(* Ange vilken datumarray som är aktuell beroende på aktuellt år *)
IF _uiYY=2017
THEN AktuellDatumArray:=Array2017;
ELSIF _uiYY=2018
THEN AktuellDatumArray:=Array2018;
ELSIF _uiYY=2019
THEN AktuellDatumArray:=Array2019;
ELSIF _uiYY=2020
THEN AktuellDatumArray:=Array2020;
ELSIF _uiYY=2021
THEN AktuellDatumArray:=Array2021;
ELSIF _uiYY=2022
THEN AktuellDatumArray:=Array2022;
ELSIF _uiYY=2023
THEN AktuellDatumArray:=Array2023;
ELSIF _uiYY=2024
THEN AktuellDatumArray:=Array2024;
ELSIF _uiYY=2025
THEN AktuellDatumArray:=Array2025;
ELSIF _uiYY=2026
THEN AktuellDatumArray:=Array2026;
ELSIF _uiYY=2027
THEN AktuellDatumArray:=Array2027;
ELSIF _uiYY=2028
THEN AktuellDatumArray:=Array2028;
ELSIF _uiYY=2029
THEN AktuellDatumArray:=Array2029;
ELSIF _uiYY=2030
THEN AktuellDatumArray:=Array2030;
ELSIF _uiYY=2031
THEN AktuellDatumArray:=Array2031;
ELSIF _uiYY=2032
THEN AktuellDatumArray:=Array2032;
ELSIF _uiYY=2033
THEN AktuellDatumArray:=Array2033;
ELSIF _uiYY=2034
THEN AktuellDatumArray:=Array2034;
ELSIF _uiYY=2035
THEN AktuellDatumArray:=Array2035;
ELSIF _uiYY=2036
THEN AktuellDatumArray:=Array2036;
ELSIF _uiYY=2037
THEN AktuellDatumArray:=Array2037;
END_IF


(* Kolla om dagens datum stämmer överens med någon av inställda helgdagar/-aftnar*)
IF _rDatum=AktuellDatumArray[1]			(*Trettondagsafton*)
OR _rDatum= AktuellDatumArray[2]			(*Skartorsdag*)
OR _rDatum=AktuellDatumArray[3]			(*Paskafton*)
OR _rDatum=AktuellDatumArray[4]			(*Valborgsmassoafton*)
OR _rDatum=AktuellDatumArray[5]			(*Pingstafton*)
OR _rDatum=AktuellDatumArray[6]			(*Midsommarafton*)
OR _rDatum=AktuellDatumArray[7]			(*AllaHelgonsAfton*)
OR _rDatum=AktuellDatumArray[8]			(*Julafton*)
OR _rDatum=AktuellDatumArray[9]			(*Nyarsafton*)
THEN bDFH:=TRUE;
ELSE bDFH:=FALSE;
END_IF

IF _rDatum=AktuellDatumArray[10]			(*Nyarsdagen*)
OR _rDatum=AktuellDatumArray[11]			(*TrettondagJul*)
OR _rDatum=AktuellDatumArray[12]			(*Langfredag*)
OR _rDatum=AktuellDatumArray[13]			(*Paskdagen*)
OR _rDatum=AktuellDatumArray[14]			(*AnnandagPask*)
OR _rDatum=AktuellDatumArray[15]			(*ForstaMaj*)
OR _rDatum=AktuellDatumArray[16]			(*KristiHimmelsfard*)
OR _rDatum=AktuellDatumArray[17]			(*Pingstdagen*)
OR _rDatum=AktuellDatumArray[18]			(*Nationaldagen*)
OR _rDatum=AktuellDatumArray[19]			(*Midsommardagen*)
OR _rDatum=AktuellDatumArray[20]			(*AllaHelgonsDag*)
OR _rDatum=AktuellDatumArray[21]			(*Juldagen*)
OR _rDatum=AktuellDatumArray[22]			(*AnnandagJul*)
THEN bHD:=TRUE;
ELSE bHD:=FALSE;
END_IF


(*Sätt larmutgång till TRUE om aktuellt årtal är större än 2037*)
IF  _uiYY>2037
THEN bLarm:=TRUE;
ELSE bLarm:=FALSE;
END_IF
END_FUNCTION_BLOCK

(* POU SYSTEM/HUS2_AS01_GT3N, CFC *)
PROGRAM HUS2_AS01_GT3N
VAR

	FilterDelay: fbDelayedAlarmMinutes;
END_VAR
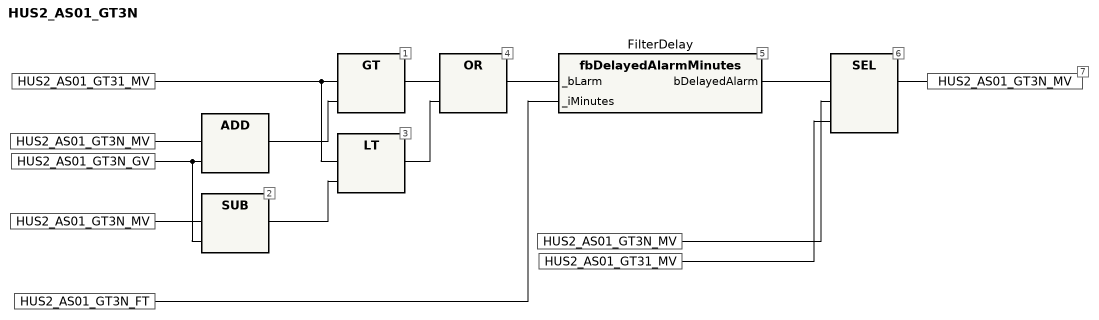
_CFC_ (* Continuous Function Chart, elements in execution order *)
#0 ADD(HUS2_AS01_GT3N_MV, HUS2_AS01_GT3N_GV)
#1 GT(HUS2_AS01_GT31_MV, #0)
#2 SUB(HUS2_AS01_GT3N_MV, HUS2_AS01_GT3N_GV)
#3 LT(HUS2_AS01_GT31_MV, #2)
#4 OR(#1, #3)
#5 FilterDelay:fbDelayedAlarmMinutes(_bLarm: #4, _iMinutes: HUS2_AS01_GT3N_FT)
#6 SEL(#5.bDelayedAlarm, HUS2_AS01_GT3N_MV, HUS2_AS01_GT31_MV)
#7 HUS2_AS01_GT3N_MV <= #6
_END_CFC_
(* the same logic as Structured Text *)
FilterDelay(_bLarm := (HUS2_AS01_GT31_MV > (HUS2_AS01_GT3N_MV + HUS2_AS01_GT3N_GV)) OR (HUS2_AS01_GT31_MV < (HUS2_AS01_GT3N_MV - HUS2_AS01_GT3N_GV)), _iMinutes := HUS2_AS01_GT3N_FT);
HUS2_AS01_GT3N_MV := SEL(FilterDelay.bDelayedAlarm, HUS2_AS01_GT3N_MV, HUS2_AS01_GT31_MV);
END_PROGRAM

(* POU SYSTEM/HUS2_AS01_SOMMARVINTER, CFC *)
PROGRAM HUS2_AS01_SOMMARVINTER

VAR
	udiIntval      : UDINT:=3600;
	udiNumOfElem   : UDINT:=72;
	lrOut             : LREAL;
	lrMax             : LREAL;
	lrMin             : LREAL;
	udiStaNumOfElem   : UDINT;

	AverageCalc: FB_HVACTimeAverage;
	ActivationDelay: TON;

	SetReset: SR;
	bVINTER_TILL: BOOL;
	TEST: BOOL := TRUE;
	TFD_VINTER: TON;
	TFD_DELAY_BER: fbINT_TO_MIN;
	FFD_VINTER: TON;
	FFD_DELAY_BER: fbINT_TO_MIN;
END_VAR
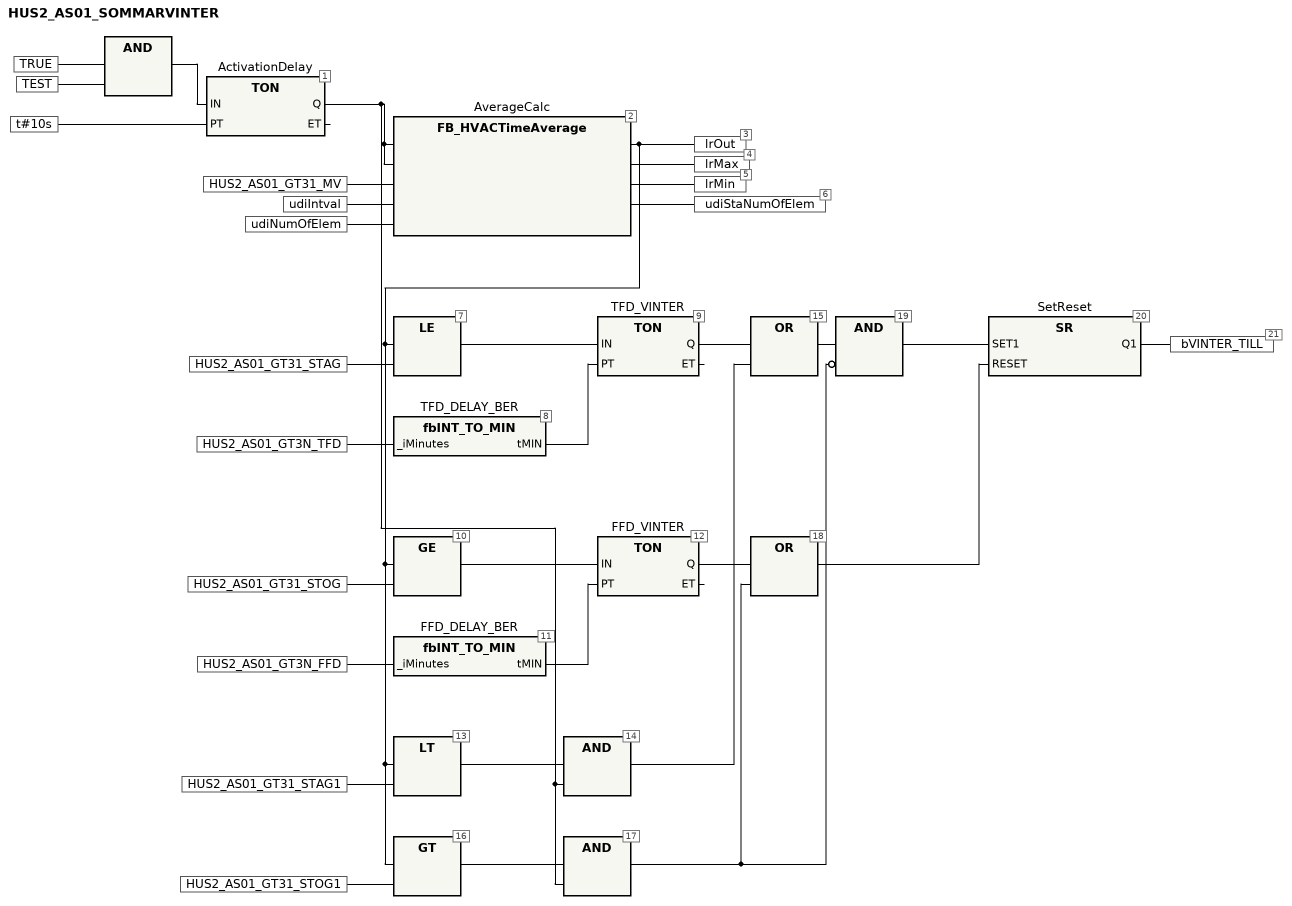
_CFC_ (* Continuous Function Chart, elements in execution order *)
#0 AND(TRUE, TEST)
#1 ActivationDelay:TON(IN: #0, PT: t#10s)
#2 AverageCalc:FB_HVACTimeAverage(#1.Q, #1.Q, HUS2_AS01_GT31_MV, udiIntval, udiNumOfElem)
#3 lrOut <= #2.out 1
#4 lrMax <= #2.out 2
#5 lrMin <= #2.out 3
#6 udiStaNumOfElem <= #2.out 4
#7 LE(#2.out 1, HUS2_AS01_GT31_STAG)
#8 TFD_DELAY_BER:fbINT_TO_MIN(_iMinutes: HUS2_AS01_GT3N_TFD)
#9 TFD_VINTER:TON(IN: #7, PT: #8.tMIN)
#10 GE(#2.out 1, HUS2_AS01_GT31_STOG)
#11 FFD_DELAY_BER:fbINT_TO_MIN(_iMinutes: HUS2_AS01_GT3N_FFD)
#12 FFD_VINTER:TON(IN: #10, PT: #11.tMIN)
#13 LT(#2.out 1, HUS2_AS01_GT31_STAG1)
#14 AND(#13, #1.Q)
#15 OR(#9.Q, #14)
#16 GT(#2.out 1, HUS2_AS01_GT31_STOG1)
#17 AND(#16, #1.Q)
#18 OR(#12.Q, #17)
#19 AND(#15, NOT #17)
#20 SetReset:SR(SET1: #19, RESET: #18)
#21 bVINTER_TILL <= #20.Q1
_END_CFC_
END_PROGRAM

(* POU xEgna Funktionsblock/fbINT_TO_MIN, CFC *)
FUNCTION_BLOCK fbINT_TO_MIN
VAR_INPUT
	_iMinutes  :INT;
END_VAR

VAR_OUTPUT
	tMIN: TIME;
END_VAR
VAR (* helpers for the ST form of the networks *)
	_t10 : TIME;
END_VAR
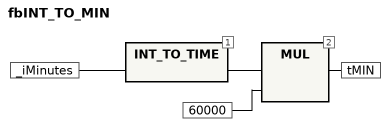
_CFC_ (* Continuous Function Chart, elements in execution order *)
#0 tMIN <= #2
#1 INT_TO_TIME(_iMinutes)
#2 MUL(#1, 60000)
_END_CFC_
(* the same logic as Structured Text *)
tMIN := _t10;
_t10 := INT_TO_TIME(_iMinutes) * 60000;
END_FUNCTION_BLOCK

(* POU SYSTEM/HUS2_AS01_LARMLAMPA, CFC *)
PROGRAM HUS2_AS01_LARMLAMPA
VAR

	BLINKALARM: FB_HVACBlink;
	ResetSet: RS;
	ACK: BOOL;
	TRIG1: R_TRIG;

	WEBPORT: BOOL;
	RESET_ACK: fbBool_Reset;
END_VAR
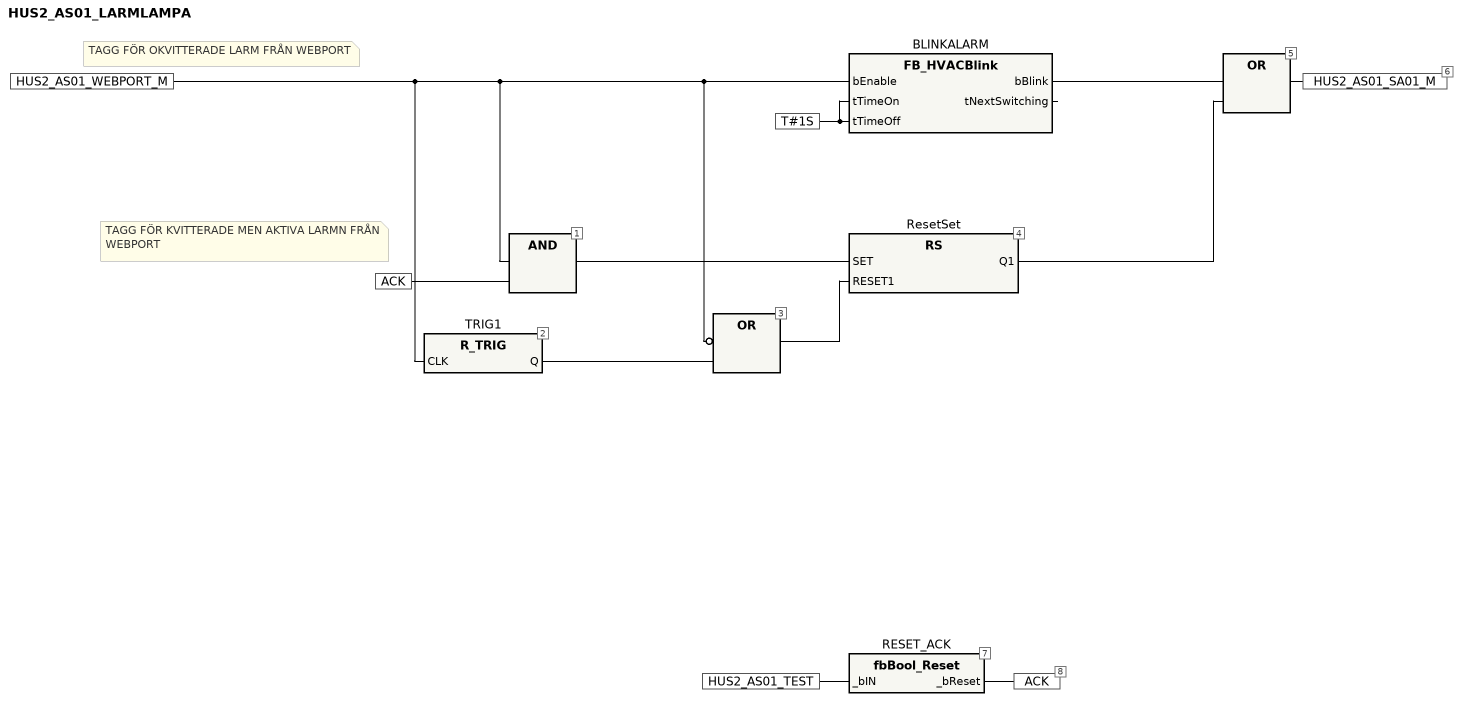
_CFC_ (* Continuous Function Chart, elements in execution order *)
(* TAGG FÖR OKVITTERADE LARM FRÅN WEBPORT *)
#0 BLINKALARM:FB_HVACBlink(bEnable: HUS2_AS01_WEBPORT_M, tTimeOn: T#1S, tTimeOff: T#1S)
#1 AND(HUS2_AS01_WEBPORT_M, ACK)
#2 TRIG1:R_TRIG(CLK: HUS2_AS01_WEBPORT_M)
#3 OR(NOT HUS2_AS01_WEBPORT_M, #2.Q)
#4 ResetSet:RS(SET: #1, RESET1: #3)
#5 OR(#0.bBlink, #4.Q1)
#6 HUS2_AS01_SA01_M <= #5
#7 RESET_ACK:fbBool_Reset(_bIN: HUS2_AS01_TEST)
#8 ACK <= #7._bReset
(* TAGG FÖR KVITTERADE MEN AKTIVA LARMN FRÅN WEBPORT *)
_END_CFC_
(* the same logic as Structured Text *)
(* TAGG FÖR OKVITTERADE LARM FRÅN WEBPORT *)
BLINKALARM(bEnable := HUS2_AS01_WEBPORT_M, tTimeOn := T#1S, tTimeOff := T#1S);
TRIG1(CLK := HUS2_AS01_WEBPORT_M);
ResetSet(SET := HUS2_AS01_WEBPORT_M AND ACK, RESET1 := NOT HUS2_AS01_WEBPORT_M OR TRIG1.Q);
HUS2_AS01_SA01_M := BLINKALARM.bBlink OR ResetSet.Q1;
RESET_ACK(_bIN := HUS2_AS01_TEST);
ACK := RESET_ACK._bReset;
(* TAGG FÖR KVITTERADE MEN AKTIVA LARMN FRÅN WEBPORT *)
END_PROGRAM

(* POU SYSTEM/Belysning/HUS2_AS01_Belysning_MAIN, CFC *)
PROGRAM HUS2_AS01_Belysning_MAIN
VAR
	LUXSTYR_BE01: fbLUX_ON_OFF;
	LUXSTYR_BE02: fbLUX_ON_OFF;
END_VAR
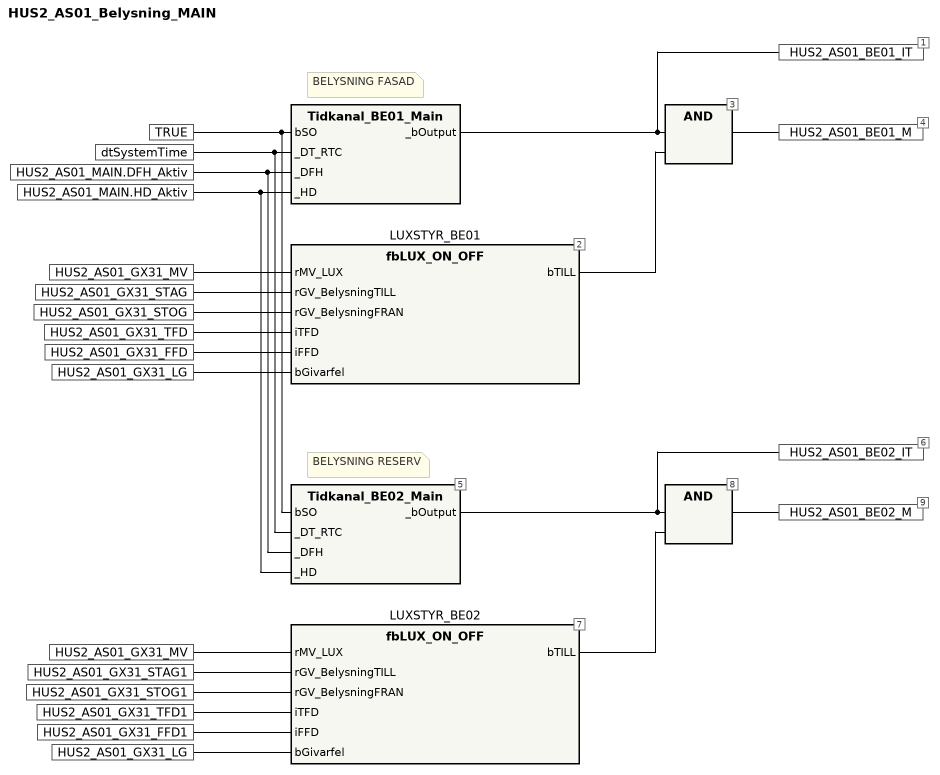
_CFC_ (* Continuous Function Chart, elements in execution order *)
(* BELYSNING FASAD *)
(* BELYSNING RESERV *)
#0 Tidkanal_BE01_Main(bSO: TRUE, _DT_RTC: dtSystemTime, _DFH: HUS2_AS01_MAIN.DFH_Aktiv, _HD: HUS2_AS01_MAIN.HD_Aktiv)
#1 HUS2_AS01_BE01_IT <= #0._bOutput
#2 LUXSTYR_BE01:fbLUX_ON_OFF(rMV_LUX: HUS2_AS01_GX31_MV, rGV_BelysningTILL: HUS2_AS01_GX31_STAG, rGV_BelysningFRAN: HUS2_AS01_GX31_STOG, iTFD: HUS2_AS01_GX31_TFD, iFFD: HUS2_AS01_GX31_FFD, bGivarfel: HUS2_AS01_GX31_LG)
#3 AND(#0._bOutput, #2.bTILL)
#4 HUS2_AS01_BE01_M <= #3
#5 Tidkanal_BE02_Main(bSO: TRUE, _DT_RTC: dtSystemTime, _DFH: HUS2_AS01_MAIN.DFH_Aktiv, _HD: HUS2_AS01_MAIN.HD_Aktiv)
#6 HUS2_AS01_BE02_IT <= #5._bOutput
#7 LUXSTYR_BE02:fbLUX_ON_OFF(rMV_LUX: HUS2_AS01_GX31_MV, rGV_BelysningTILL: HUS2_AS01_GX31_STAG1, rGV_BelysningFRAN: HUS2_AS01_GX31_STOG1, iTFD: HUS2_AS01_GX31_TFD1, iFFD: HUS2_AS01_GX31_FFD1, bGivarfel: HUS2_AS01_GX31_LG)
#8 AND(#5._bOutput, #7.bTILL)
#9 HUS2_AS01_BE02_M <= #8
_END_CFC_
(* the same logic as Structured Text *)
(* BELYSNING FASAD *)
(* BELYSNING RESERV *)
Tidkanal_BE01_Main(bSO := TRUE, _DT_RTC := dtSystemTime, _DFH := HUS2_AS01_MAIN.DFH_Aktiv, _HD := HUS2_AS01_MAIN.HD_Aktiv);
HUS2_AS01_BE01_IT := Tidkanal_BE01_Main._bOutput;
LUXSTYR_BE01(rMV_LUX := HUS2_AS01_GX31_MV, rGV_BelysningTILL := HUS2_AS01_GX31_STAG, rGV_BelysningFRAN := HUS2_AS01_GX31_STOG, iTFD := HUS2_AS01_GX31_TFD, iFFD := HUS2_AS01_GX31_FFD, bGivarfel := HUS2_AS01_GX31_LG);
HUS2_AS01_BE01_M := Tidkanal_BE01_Main._bOutput AND LUXSTYR_BE01.bTILL;
Tidkanal_BE02_Main(bSO := TRUE, _DT_RTC := dtSystemTime, _DFH := HUS2_AS01_MAIN.DFH_Aktiv, _HD := HUS2_AS01_MAIN.HD_Aktiv);
HUS2_AS01_BE02_IT := Tidkanal_BE02_Main._bOutput;
LUXSTYR_BE02(rMV_LUX := HUS2_AS01_GX31_MV, rGV_BelysningTILL := HUS2_AS01_GX31_STAG1, rGV_BelysningFRAN := HUS2_AS01_GX31_STOG1, iTFD := HUS2_AS01_GX31_TFD1, iFFD := HUS2_AS01_GX31_FFD1, bGivarfel := HUS2_AS01_GX31_LG);
HUS2_AS01_BE02_M := Tidkanal_BE02_Main._bOutput AND LUXSTYR_BE02.bTILL;
END_PROGRAM

(* POU xEgna Funktionsblock/fbLUX_ON_OFF, CFC *)
FUNCTION_BLOCK fbLUX_ON_OFF

VAR_INPUT
	rMV_LUX					: REAL;
	rGV_BelysningTILL		: REAL;
	rGV_BelysningFRAN		: REAL;
	iTFD						: INT;
	iFFD						: INT;
	bGivarfel					: BOOL;
END_VAR
VAR
	DelayON: TON;
	DelayOFF: TON;
	SETRESET: SR;
END_VAR
VAR_OUTPUT
	bTILL: BOOL;
END_VAR
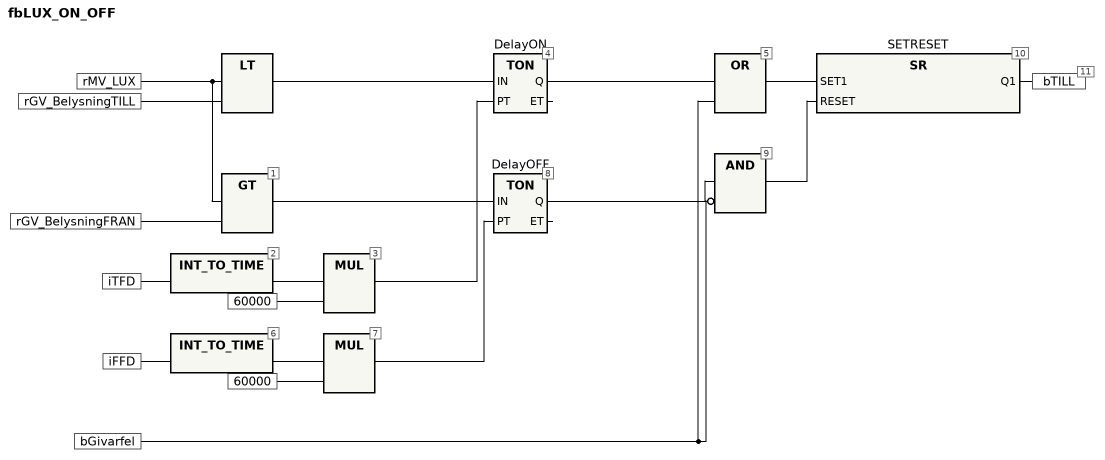
_CFC_ (* Continuous Function Chart, elements in execution order *)
#0 LT(rMV_LUX, rGV_BelysningTILL)
#1 GT(rMV_LUX, rGV_BelysningFRAN)
#2 INT_TO_TIME(iTFD)
#3 MUL(#2, 60000)
#4 DelayON:TON(IN: #0, PT: #3)
#5 OR(#4.Q, bGivarfel)
#6 INT_TO_TIME(iFFD)
#7 MUL(#6, 60000)
#8 DelayOFF:TON(IN: #1, PT: #7)
#9 AND(#8.Q, NOT bGivarfel)
#10 SETRESET:SR(SET1: #5, RESET: #9)
#11 bTILL <= #10.Q1
_END_CFC_
(* the same logic as Structured Text *)
DelayON(IN := rMV_LUX < rGV_BelysningTILL, PT := INT_TO_TIME(iTFD) * 60000);
DelayOFF(IN := rMV_LUX > rGV_BelysningFRAN, PT := INT_TO_TIME(iFFD) * 60000);
SETRESET(SET1 := DelayON.Q OR bGivarfel, RESET := DelayOFF.Q AND NOT bGivarfel);
bTILL := SETRESET.Q1;
END_FUNCTION_BLOCK

(* POU SYSTEM/Belysning/BE01/Tidkanal_BE01_Main, CFC *)
PROGRAM Tidkanal_BE01_Main

VAR_INPUT
	bSO: BOOL;
	_DT_RTC	:DT;
	_DFH :BOOL;
	_HD:BOOL;

END_VAR


VAR
	AUTO_MAN: fbManualOverride;

	OffDelayTK: TOF;
END_VAR

VAR_OUTPUT
	_bOutput:BOOL;

END_VAR
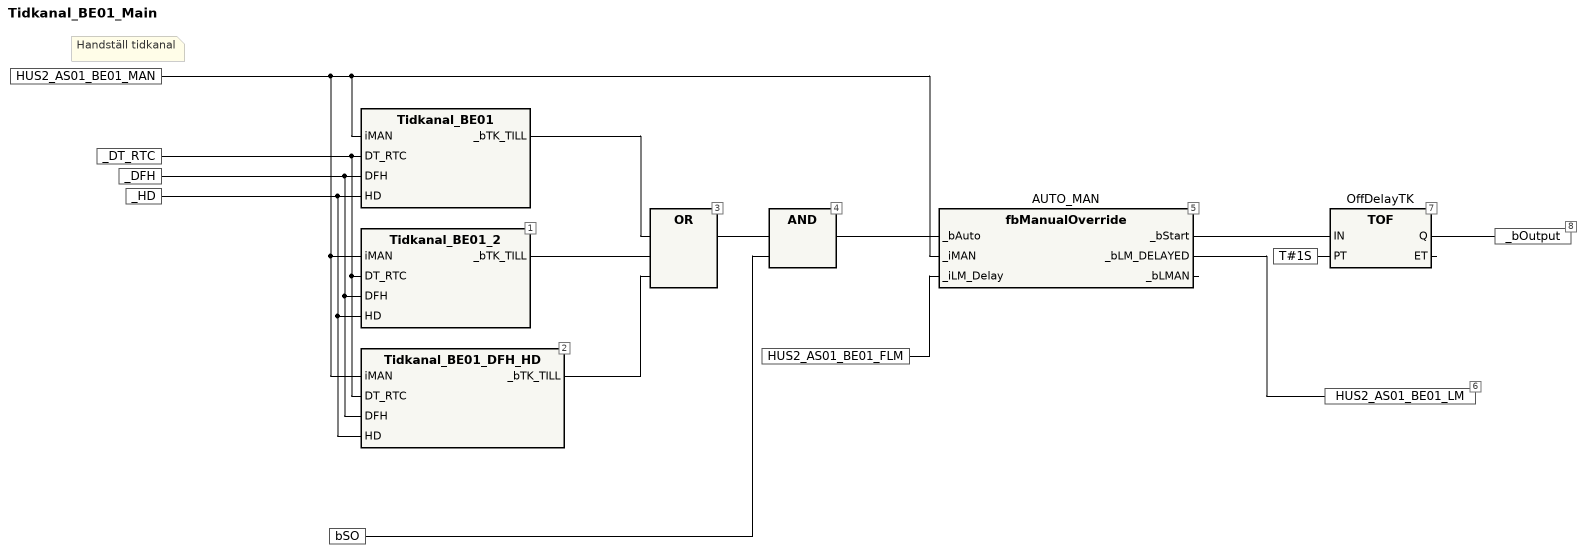
_CFC_ (* Continuous Function Chart, elements in execution order *)
(* Handställ tidkanal *)
#0 Tidkanal_BE01(iMAN: HUS2_AS01_BE01_MAN, DT_RTC: _DT_RTC, DFH: _DFH, HD: _HD)
#1 Tidkanal_BE01_2(iMAN: HUS2_AS01_BE01_MAN, DT_RTC: _DT_RTC, DFH: _DFH, HD: _HD)
#2 Tidkanal_BE01_DFH_HD(iMAN: HUS2_AS01_BE01_MAN, DT_RTC: _DT_RTC, DFH: _DFH, HD: _HD)
#3 OR(#0._bTK_TILL, #1._bTK_TILL, #2._bTK_TILL)
#4 AND(#3, bSO)
#5 AUTO_MAN:fbManualOverride(_bAuto: #4, _iMAN: HUS2_AS01_BE01_MAN, _iLM_Delay: HUS2_AS01_BE01_FLM)
#6 HUS2_AS01_BE01_LM <= #5._bLM_DELAYED
#7 OffDelayTK:TOF(IN: #5._bStart, PT: T#1S)
#8 _bOutput <= #7.Q
_END_CFC_
(* the same logic as Structured Text *)
(* Handställ tidkanal *)
Tidkanal_BE01(iMAN := HUS2_AS01_BE01_MAN, DT_RTC := _DT_RTC, DFH := _DFH, HD := _HD);
Tidkanal_BE01_2(iMAN := HUS2_AS01_BE01_MAN, DT_RTC := _DT_RTC, DFH := _DFH, HD := _HD);
Tidkanal_BE01_DFH_HD(iMAN := HUS2_AS01_BE01_MAN, DT_RTC := _DT_RTC, DFH := _DFH, HD := _HD);
AUTO_MAN(_bAuto := (Tidkanal_BE01._bTK_TILL OR Tidkanal_BE01_2._bTK_TILL OR Tidkanal_BE01_DFH_HD._bTK_TILL) AND bSO, _iMAN := HUS2_AS01_BE01_MAN, _iLM_Delay := HUS2_AS01_BE01_FLM);
HUS2_AS01_BE01_LM := AUTO_MAN._bLM_DELAYED;
OffDelayTK(IN := AUTO_MAN._bStart, PT := T#1S);
_bOutput := OffDelayTK.Q;
END_PROGRAM

(* POU xEgna Funktionsblock/fbManualOverride, CFC *)
FUNCTION_BLOCK fbManualOverride
VAR_INPUT
	_bAuto:BOOL;
	_iMAN: INT;
	_iLM_Delay: INT;
END_VAR
VAR_OUTPUT
	_bStart: BOOL;
	_bLM_DELAYED: BOOL;
	_bLMAN: BOOL;
END_VAR
VAR
	LM_DELAY: fbDelayedAlarmMinutes;
	OFF_DELAY: TOF;
END_VAR
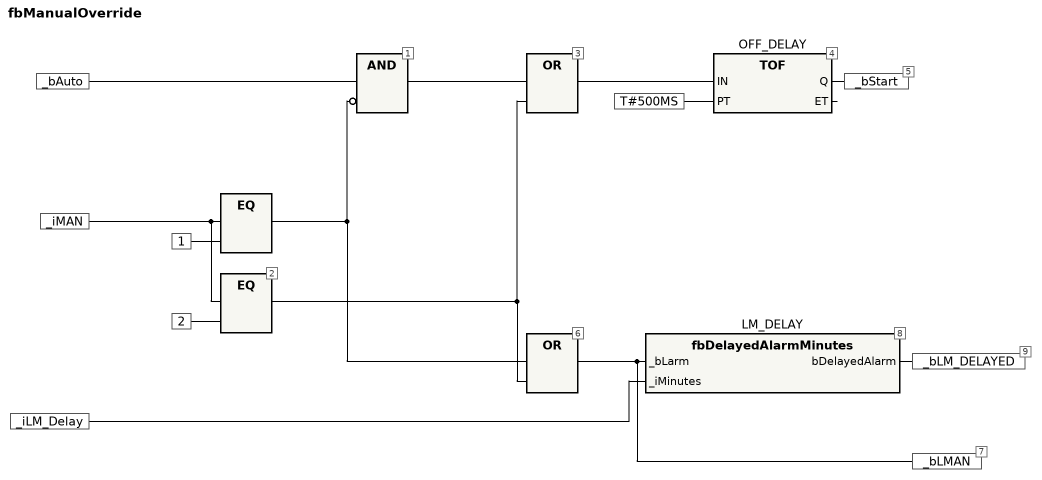
_CFC_ (* Continuous Function Chart, elements in execution order *)
#0 EQ(_iMAN, 1)
#1 AND(_bAuto, NOT #0)
#2 EQ(_iMAN, 2)
#3 OR(#1, #2)
#4 OFF_DELAY:TOF(IN: #3, PT: T#500MS)
#5 _bStart <= #4.Q
#6 OR(#0, #2)
#7 _bLMAN <= #6
#8 LM_DELAY:fbDelayedAlarmMinutes(_bLarm: #6, _iMinutes: _iLM_Delay)
#9 _bLM_DELAYED <= #8.bDelayedAlarm
_END_CFC_
(* the same logic as Structured Text *)
OFF_DELAY(IN := (_bAuto AND NOT (_iMAN = 1)) OR (_iMAN = 2), PT := T#500MS);
_bStart := OFF_DELAY.Q;
_bLMAN := (_iMAN = 1) OR (_iMAN = 2);
LM_DELAY(_bLarm := (_iMAN = 1) OR (_iMAN = 2), _iMinutes := _iLM_Delay);
_bLM_DELAYED := LM_DELAY.bDelayedAlarm;
END_FUNCTION_BLOCK

(* POU SYSTEM/Belysning/BE01/Tidkanal_BE01, FAI *)
PROGRAM Tidkanal_BE01

VAR

(****************************************  weekly time switch *********************************************************************************************************************)
	fbWeeklyTimeSwitch		:FB_HVACScheduler7ch;
	_eDST					:E_HVACDataSecurityType :=1;
	SetDefaultTimeSwitch: BOOL := FALSE;
	_uiOffsetBefore			:UINT;  (* the switch-on time is brought forward by this number of minutes *)
	_arrTimeChannel 			:ARRAY[1..7] OF ST_HVACTimeChannel;(*
							    ST_HVACTimeChannel :
							    uiOn_hh			: UINT;
							    uiOn_mm		: UINT;
							    uiOn_ss			: UINT;
							    uiOff_hh			: UINT; 
							    uiOff_mm			: UINT;
							    uiOff_ss			: UINT;
							    bEnable			: BOOL;
							    bAllDays			: BOOL;
							    bMonday			: BOOL;
							    bTuesday		: BOOL;
							    bWednesday		: BOOL;
							    bThursday		: BOOL;
							    bFriday			: BOOL;
							    bSaturday		: BOOL;
							    bSunday			: BOOL;
							    bResetAfterOn	: BOOL;
							    bQ				: BOOL; *)

	_bWeeklyClock_EdgeOn		:BOOL;(* Is TRUE for one PLC cycle after bOutput switches on *)
	_bWeeklyClock_EdgeOff		:BOOL;(* Is TRUE for one PLC cycle after bOutput switches off *)
	_tWeeklyTime_NextOn		:TIME;(* Time until the next switch-on of the time switch program. Maximum value 10080 minutes (1 week) *)
	_tWeeklyTime_NextOff		:TIME;(* Time until the next switch-off of the time switch program. Maximum forecast until midnight *)
	_bWeeklyTime_FP			:BOOL;(* fault parameter recognized *)



	_bReset_Local				:BOOL;
	_bSetDefault_Local: BOOL;

	fbSCADATime1:		FB_TimeToSCADA_1_0;
	fbSCADATime2:		FB_TimeToSCADA_1_0;
	fbSCADATime3:		FB_TimeToSCADA_1_0;
	fbSCADATime4:		FB_TimeToSCADA_1_0;
	fbSCADATime5:		FB_TimeToSCADA_1_0;
	fbSCADATime6:		FB_TimeToSCADA_1_0;
	fbSCADATime7:		FB_TimeToSCADA_1_0;






END_VAR


VAR_INPUT
	iMAN				:INT;
	DT_RTC			:DT;
	DFH 				:BOOL;
	HD					:BOOL;

END_VAR

VAR_OUTPUT
	_bTK_TILL		:BOOL;

END_VAR
(* body not read: cfc101 *)
END_PROGRAM

(* POU xEgna Funktionsblock/Time_to_SCADA/FB_TimeToSCADA_1_0, ST *)
(*
Lib: TCHVAC.LIB
*)

FUNCTION_BLOCK FB_TimeToSCADA_1_0

VAR_INPUT
END_VAR

VAR_IN_OUT
	_iCitect_OnTime:		INT;		(*Time On from HMI*)
	_iCitect_OffTime:		INT;		(*Time Off from HMI*)
END_VAR
VAR_OUTPUT
	_uiOnTime_hh:		UINT;		(*Hours for on time*)
	_uiOnTime_mm:		UINT;		(*Minutes for on time*)
	_uiOffTime_hh:		UINT;		(*Hours for off time*)
	_uiOffTime_mm:		UINT;		(*Minutes for off time*)
	_bEnableTimeCh:		BOOL;		(*Enable timechannel*)
END_VAR
VAR
	iNowOn:				INT;		(*Temp var for on time*)
	iNowOff:				INT;		(*Temp var for off time*)
	fbSaveOnTime:		FB_HVACPersistent_Int;
	fbSaveOffTime:		FB_HVACPersistent_Int;
END_VAR

(*
	This FB converts hmi time from Citect to HVAC TimeChannel
	the input time is an integer. i.e Time 15:46 = _iCitect_OnTime 1546. Then
	the our and minute is extracted to the HVAC time. 
	No error handling if time is not in the appropriate range.
	Maybe the persistent data handling for the TC needs to be disabled
*)
(*Find out if we have some time set, then enable the output*)
IF
_iCitect_OffTime <> _iCitect_OnTime
THEN
(*Get the on time*)
iNowOn := _iCitect_OnTime;
(*Get hour*)
_uiOnTime_hh := iNowOn / 100;
(*Get minute*)
_uiOnTime_mm := iNowOn - ( _uiOnTime_hh * 100);

(*Get the off time*)
iNowOff := _iCitect_OffTime;
(*Get hour*)
_uiOffTime_hh := iNowOff / 100;
(*Get minute*)
_uiOffTime_mm := iNowOff - ( _uiOffTime_hh * 100);
	_bEnableTimeCh := TRUE;
ELSIF
_iCitect_OffTime=2359 AND _iCitect_OnTime=2359
OR
_iCitect_OffTime=2400 AND _iCitect_OnTime=0000
THEN
	_uiOnTime_hh:=0;
	_uiOnTime_mm:=0;
	_uiOffTime_hh:=0;
	_uiOffTime_mm:=0;
	_bEnableTimeCh:=0;
	_bEnableTimeCh := TRUE;
ELSE
	_bEnableTimeCh := FALSE;
END_IF


(*Save the on/off time data persistent*)
fbSaveOnTime(bSetDefault:= , iVar_Default:= , iVar:= _iCitect_OnTime );
fbSaveOffTime(bSetDefault:= , iVar_Default:= , iVar:= _iCitect_OffTime );
END_FUNCTION_BLOCK

(* POU SYSTEM/Belysning/BE01/Tidkanal_BE01_2, FAI *)
PROGRAM Tidkanal_BE01_2

VAR

(****************************************  weekly time switch *********************************************************************************************************************)
	fbWeeklyTimeSwitch		:FB_HVACScheduler7ch;
	_eDST					:E_HVACDataSecurityType :=1;
	SetDefaultTimeSwitch: BOOL := FALSE;
	_uiOffsetBefore			:UINT;  (* the switch-on time is brought forward by this number of minutes *)
	_arrTimeChannel 			:ARRAY[1..7] OF ST_HVACTimeChannel;(*
							    ST_HVACTimeChannel :
							    uiOn_hh			: UINT;
							    uiOn_mm		: UINT;
							    uiOn_ss			: UINT;
							    uiOff_hh			: UINT; 
							    uiOff_mm			: UINT;
							    uiOff_ss			: UINT;
							    bEnable			: BOOL;
							    bAllDays			: BOOL;
							    bMonday			: BOOL;
							    bTuesday		: BOOL;
							    bWednesday		: BOOL;
							    bThursday		: BOOL;
							    bFriday			: BOOL;
							    bSaturday		: BOOL;
							    bSunday			: BOOL;
							    bResetAfterOn	: BOOL;
							    bQ				: BOOL; *)

	_bWeeklyClock_EdgeOn		:BOOL;(* Is TRUE for one PLC cycle after bOutput switches on *)
	_bWeeklyClock_EdgeOff		:BOOL;(* Is TRUE for one PLC cycle after bOutput switches off *)
	_tWeeklyTime_NextOn		:TIME;(* Time until the next switch-on of the time switch program. Maximum value 10080 minutes (1 week) *)
	_tWeeklyTime_NextOff		:TIME;(* Time until the next switch-off of the time switch program. Maximum forecast until midnight *)
	_bWeeklyTime_FP			:BOOL;(* fault parameter recognized *)



	_bReset_Local				:BOOL;
	_bSetDefault_Local: BOOL;

	fbSCADATime1:		FB_TimeToSCADA_1_0;
	fbSCADATime2:		FB_TimeToSCADA_1_0;
	fbSCADATime3:		FB_TimeToSCADA_1_0;
	fbSCADATime4:		FB_TimeToSCADA_1_0;
	fbSCADATime5:		FB_TimeToSCADA_1_0;
	fbSCADATime6:		FB_TimeToSCADA_1_0;
	fbSCADATime7:		FB_TimeToSCADA_1_0;






END_VAR


VAR_INPUT
	iMAN				:INT;
	DT_RTC			:DT;
	DFH 				:BOOL;
	HD					:BOOL;

END_VAR

VAR_OUTPUT
	_bTK_TILL		:BOOL;

END_VAR
(* body not read: cfc101 *)
END_PROGRAM

(* POU SYSTEM/Belysning/BE01/Tidkanal_BE01_DFH_HD, FAI *)
PROGRAM Tidkanal_BE01_DFH_HD

VAR

(****************************************  weekly time switch *********************************************************************************************************************)
	fbWeeklyTimeSwitch		:FB_HVACScheduler7ch;
	_eDST					:E_HVACDataSecurityType :=1;
	SetDefaultTimeSwitch: BOOL := FALSE;
	_uiOffsetBefore			:UINT;  (* the switch-on time is brought forward by this number of minutes *)
	_arrTimeChannel 			:ARRAY[1..7] OF ST_HVACTimeChannel;(*
							    ST_HVACTimeChannel :
							    uiOn_hh			: UINT;
							    uiOn_mm		: UINT;
							    uiOn_ss			: UINT;
							    uiOff_hh			: UINT; 
							    uiOff_mm			: UINT;
							    uiOff_ss			: UINT;
							    bEnable			: BOOL;
							    bAllDays			: BOOL;
							    bMonday			: BOOL;
							    bTuesday		: BOOL;
							    bWednesday		: BOOL;
							    bThursday		: BOOL;
							    bFriday			: BOOL;
							    bSaturday		: BOOL;
							    bSunday			: BOOL;
							    bResetAfterOn	: BOOL;
							    bQ				: BOOL; *)

	_bWeeklyClock_EdgeOn		:BOOL;(* Is TRUE for one PLC cycle after bOutput switches on *)
	_bWeeklyClock_EdgeOff		:BOOL;(* Is TRUE for one PLC cycle after bOutput switches off *)
	_tWeeklyTime_NextOn		:TIME;(* Time until the next switch-on of the time switch program. Maximum value 10080 minutes (1 week) *)
	_tWeeklyTime_NextOff		:TIME;(* Time until the next switch-off of the time switch program. Maximum forecast until midnight *)
	_bWeeklyTime_FP			:BOOL;(* fault parameter recognized *)



	_bReset_Local				:BOOL;
	_bSetDefault_Local: BOOL;

	fbSCADATime1:		FB_TimeToSCADA_1_0;
	fbSCADATime2:		FB_TimeToSCADA_1_0;
	fbSCADATime3:		FB_TimeToSCADA_1_0;
	fbSCADATime4:		FB_TimeToSCADA_1_0;
	fbSCADATime5:		FB_TimeToSCADA_1_0;
	fbSCADATime6:		FB_TimeToSCADA_1_0;
	fbSCADATime7:		FB_TimeToSCADA_1_0;






END_VAR


VAR_INPUT
	iMAN				:INT;
	DT_RTC			:DT;
	DFH 				:BOOL;
	HD					:BOOL;

END_VAR

VAR_OUTPUT
	_bTK_TILL		:BOOL;

END_VAR
(* body not read: cfc101 *)
END_PROGRAM

(* POU SYSTEM/Belysning/BE02/Tidkanal_BE02_Main, CFC *)
PROGRAM Tidkanal_BE02_Main

VAR_INPUT
	bSO: BOOL;
	_DT_RTC	:DT;
	_DFH :BOOL;
	_HD:BOOL;

END_VAR


VAR
	AUTO_MAN: fbManualOverride;

	OffDelayTK: TOF;
END_VAR

VAR_OUTPUT
	_bOutput:BOOL;

END_VAR
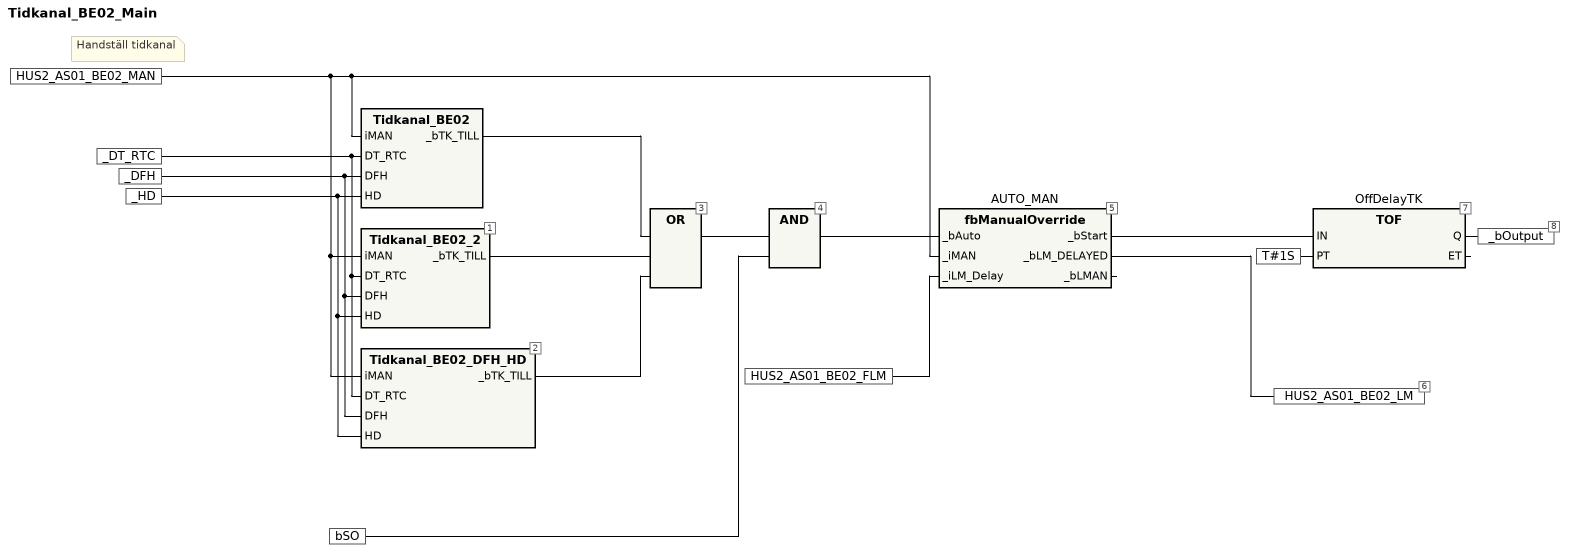
_CFC_ (* Continuous Function Chart, elements in execution order *)
(* Handställ tidkanal *)
#0 Tidkanal_BE02(iMAN: HUS2_AS01_BE02_MAN, DT_RTC: _DT_RTC, DFH: _DFH, HD: _HD)
#1 Tidkanal_BE02_2(iMAN: HUS2_AS01_BE02_MAN, DT_RTC: _DT_RTC, DFH: _DFH, HD: _HD)
#2 Tidkanal_BE02_DFH_HD(iMAN: HUS2_AS01_BE02_MAN, DT_RTC: _DT_RTC, DFH: _DFH, HD: _HD)
#3 OR(#0._bTK_TILL, #1._bTK_TILL, #2._bTK_TILL)
#4 AND(#3, bSO)
#5 AUTO_MAN:fbManualOverride(_bAuto: #4, _iMAN: HUS2_AS01_BE02_MAN, _iLM_Delay: HUS2_AS01_BE02_FLM)
#6 HUS2_AS01_BE02_LM <= #5._bLM_DELAYED
#7 OffDelayTK:TOF(IN: #5._bStart, PT: T#1S)
#8 _bOutput <= #7.Q
_END_CFC_
(* the same logic as Structured Text *)
(* Handställ tidkanal *)
Tidkanal_BE02(iMAN := HUS2_AS01_BE02_MAN, DT_RTC := _DT_RTC, DFH := _DFH, HD := _HD);
Tidkanal_BE02_2(iMAN := HUS2_AS01_BE02_MAN, DT_RTC := _DT_RTC, DFH := _DFH, HD := _HD);
Tidkanal_BE02_DFH_HD(iMAN := HUS2_AS01_BE02_MAN, DT_RTC := _DT_RTC, DFH := _DFH, HD := _HD);
AUTO_MAN(_bAuto := (Tidkanal_BE02._bTK_TILL OR Tidkanal_BE02_2._bTK_TILL OR Tidkanal_BE02_DFH_HD._bTK_TILL) AND bSO, _iMAN := HUS2_AS01_BE02_MAN, _iLM_Delay := HUS2_AS01_BE02_FLM);
HUS2_AS01_BE02_LM := AUTO_MAN._bLM_DELAYED;
OffDelayTK(IN := AUTO_MAN._bStart, PT := T#1S);
_bOutput := OffDelayTK.Q;
END_PROGRAM

(* POU SYSTEM/Belysning/BE02/Tidkanal_BE02, FAI *)
PROGRAM Tidkanal_BE02

VAR

(****************************************  weekly time switch *********************************************************************************************************************)
	fbWeeklyTimeSwitch		:FB_HVACScheduler7ch;
	_eDST					:E_HVACDataSecurityType :=1;
	SetDefaultTimeSwitch: BOOL := FALSE;
	_uiOffsetBefore			:UINT;  (* the switch-on time is brought forward by this number of minutes *)
	_arrTimeChannel 			:ARRAY[1..7] OF ST_HVACTimeChannel;(*
							    ST_HVACTimeChannel :
							    uiOn_hh			: UINT;
							    uiOn_mm		: UINT;
							    uiOn_ss			: UINT;
							    uiOff_hh			: UINT; 
							    uiOff_mm			: UINT;
							    uiOff_ss			: UINT;
							    bEnable			: BOOL;
							    bAllDays			: BOOL;
							    bMonday			: BOOL;
							    bTuesday		: BOOL;
							    bWednesday		: BOOL;
							    bThursday		: BOOL;
							    bFriday			: BOOL;
							    bSaturday		: BOOL;
							    bSunday			: BOOL;
							    bResetAfterOn	: BOOL;
							    bQ				: BOOL; *)

	_bWeeklyClock_EdgeOn		:BOOL;(* Is TRUE for one PLC cycle after bOutput switches on *)
	_bWeeklyClock_EdgeOff		:BOOL;(* Is TRUE for one PLC cycle after bOutput switches off *)
	_tWeeklyTime_NextOn		:TIME;(* Time until the next switch-on of the time switch program. Maximum value 10080 minutes (1 week) *)
	_tWeeklyTime_NextOff		:TIME;(* Time until the next switch-off of the time switch program. Maximum forecast until midnight *)
	_bWeeklyTime_FP			:BOOL;(* fault parameter recognized *)



	_bReset_Local				:BOOL;
	_bSetDefault_Local: BOOL;

	fbSCADATime1:		FB_TimeToSCADA_1_0;
	fbSCADATime2:		FB_TimeToSCADA_1_0;
	fbSCADATime3:		FB_TimeToSCADA_1_0;
	fbSCADATime4:		FB_TimeToSCADA_1_0;
	fbSCADATime5:		FB_TimeToSCADA_1_0;
	fbSCADATime6:		FB_TimeToSCADA_1_0;
	fbSCADATime7:		FB_TimeToSCADA_1_0;






END_VAR


VAR_INPUT
	iMAN				:INT;
	DT_RTC			:DT;
	DFH 				:BOOL;
	HD					:BOOL;

END_VAR

VAR_OUTPUT
	_bTK_TILL		:BOOL;

END_VAR
(* body not read: cfc101 *)
END_PROGRAM

(* POU SYSTEM/Belysning/BE02/Tidkanal_BE02_2, FAI *)
PROGRAM Tidkanal_BE02_2

VAR

(****************************************  weekly time switch *********************************************************************************************************************)
	fbWeeklyTimeSwitch		:FB_HVACScheduler7ch;
	_eDST					:E_HVACDataSecurityType :=1;
	SetDefaultTimeSwitch: BOOL := FALSE;
	_uiOffsetBefore			:UINT;  (* the switch-on time is brought forward by this number of minutes *)
	_arrTimeChannel 			:ARRAY[1..7] OF ST_HVACTimeChannel;(*
							    ST_HVACTimeChannel :
							    uiOn_hh			: UINT;
							    uiOn_mm		: UINT;
							    uiOn_ss			: UINT;
							    uiOff_hh			: UINT; 
							    uiOff_mm			: UINT;
							    uiOff_ss			: UINT;
							    bEnable			: BOOL;
							    bAllDays			: BOOL;
							    bMonday			: BOOL;
							    bTuesday		: BOOL;
							    bWednesday		: BOOL;
							    bThursday		: BOOL;
							    bFriday			: BOOL;
							    bSaturday		: BOOL;
							    bSunday			: BOOL;
							    bResetAfterOn	: BOOL;
							    bQ				: BOOL; *)

	_bWeeklyClock_EdgeOn		:BOOL;(* Is TRUE for one PLC cycle after bOutput switches on *)
	_bWeeklyClock_EdgeOff		:BOOL;(* Is TRUE for one PLC cycle after bOutput switches off *)
	_tWeeklyTime_NextOn		:TIME;(* Time until the next switch-on of the time switch program. Maximum value 10080 minutes (1 week) *)
	_tWeeklyTime_NextOff		:TIME;(* Time until the next switch-off of the time switch program. Maximum forecast until midnight *)
	_bWeeklyTime_FP			:BOOL;(* fault parameter recognized *)



	_bReset_Local				:BOOL;
	_bSetDefault_Local: BOOL;

	fbSCADATime1:		FB_TimeToSCADA_1_0;
	fbSCADATime2:		FB_TimeToSCADA_1_0;
	fbSCADATime3:		FB_TimeToSCADA_1_0;
	fbSCADATime4:		FB_TimeToSCADA_1_0;
	fbSCADATime5:		FB_TimeToSCADA_1_0;
	fbSCADATime6:		FB_TimeToSCADA_1_0;
	fbSCADATime7:		FB_TimeToSCADA_1_0;






END_VAR


VAR_INPUT
	iMAN				:INT;
	DT_RTC			:DT;
	DFH 				:BOOL;
	HD					:BOOL;

END_VAR

VAR_OUTPUT
	_bTK_TILL		:BOOL;

END_VAR
(* body not read: cfc101 *)
END_PROGRAM

(* POU SYSTEM/Belysning/BE02/Tidkanal_BE02_DFH_HD, FAI *)
PROGRAM Tidkanal_BE02_DFH_HD

VAR

(****************************************  weekly time switch *********************************************************************************************************************)
	fbWeeklyTimeSwitch		:FB_HVACScheduler7ch;
	_eDST					:E_HVACDataSecurityType :=1;
	SetDefaultTimeSwitch: BOOL := FALSE;
	_uiOffsetBefore			:UINT;  (* the switch-on time is brought forward by this number of minutes *)
	_arrTimeChannel 			:ARRAY[1..7] OF ST_HVACTimeChannel;(*
							    ST_HVACTimeChannel :
							    uiOn_hh			: UINT;
							    uiOn_mm		: UINT;
							    uiOn_ss			: UINT;
							    uiOff_hh			: UINT; 
							    uiOff_mm			: UINT;
							    uiOff_ss			: UINT;
							    bEnable			: BOOL;
							    bAllDays			: BOOL;
							    bMonday			: BOOL;
							    bTuesday		: BOOL;
							    bWednesday		: BOOL;
							    bThursday		: BOOL;
							    bFriday			: BOOL;
							    bSaturday		: BOOL;
							    bSunday			: BOOL;
							    bResetAfterOn	: BOOL;
							    bQ				: BOOL; *)

	_bWeeklyClock_EdgeOn		:BOOL;(* Is TRUE for one PLC cycle after bOutput switches on *)
	_bWeeklyClock_EdgeOff		:BOOL;(* Is TRUE for one PLC cycle after bOutput switches off *)
	_tWeeklyTime_NextOn		:TIME;(* Time until the next switch-on of the time switch program. Maximum value 10080 minutes (1 week) *)
	_tWeeklyTime_NextOff		:TIME;(* Time until the next switch-off of the time switch program. Maximum forecast until midnight *)
	_bWeeklyTime_FP			:BOOL;(* fault parameter recognized *)



	_bReset_Local				:BOOL;
	_bSetDefault_Local: BOOL;

	fbSCADATime1:		FB_TimeToSCADA_1_0;
	fbSCADATime2:		FB_TimeToSCADA_1_0;
	fbSCADATime3:		FB_TimeToSCADA_1_0;
	fbSCADATime4:		FB_TimeToSCADA_1_0;
	fbSCADATime5:		FB_TimeToSCADA_1_0;
	fbSCADATime6:		FB_TimeToSCADA_1_0;
	fbSCADATime7:		FB_TimeToSCADA_1_0;






END_VAR


VAR_INPUT
	iMAN				:INT;
	DT_RTC			:DT;
	DFH 				:BOOL;
	HD					:BOOL;

END_VAR

VAR_OUTPUT
	_bTK_TILL		:BOOL;

END_VAR
(* body not read: cfc101 *)
END_PROGRAM

(* POU SYSTEM/Motionering/TK01_MOTION/HUS2_AS01_TK01_MOTION, CFC *)
PROGRAM HUS2_AS01_TK01_MOTION

VAR
	AUTO_MAN: fbManualOverride;

END_VAR
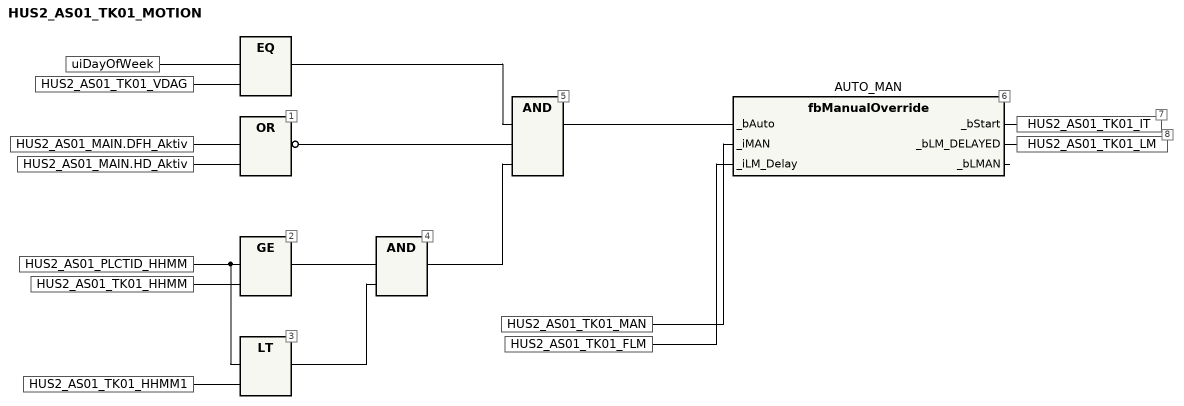
_CFC_ (* Continuous Function Chart, elements in execution order *)
#0 EQ(uiDayOfWeek, HUS2_AS01_TK01_VDAG)
#1 OR(HUS2_AS01_MAIN.DFH_Aktiv, HUS2_AS01_MAIN.HD_Aktiv)
#2 GE(HUS2_AS01_PLCTID_HHMM, HUS2_AS01_TK01_HHMM)
#3 LT(HUS2_AS01_PLCTID_HHMM, HUS2_AS01_TK01_HHMM1)
#4 AND(#2, #3)
#5 AND(#0, NOT #1, #4)
#6 AUTO_MAN:fbManualOverride(_bAuto: #5, _iMAN: HUS2_AS01_TK01_MAN, _iLM_Delay: HUS2_AS01_TK01_FLM)
#7 HUS2_AS01_TK01_IT <= #6._bStart
#8 HUS2_AS01_TK01_LM <= #6._bLM_DELAYED
_END_CFC_
(* the same logic as Structured Text *)
AUTO_MAN(_bAuto := (uiDayOfWeek = HUS2_AS01_TK01_VDAG) AND NOT (HUS2_AS01_MAIN.DFH_Aktiv OR HUS2_AS01_MAIN.HD_Aktiv) AND ((HUS2_AS01_PLCTID_HHMM >= HUS2_AS01_TK01_HHMM) AND (HUS2_AS01_PLCTID_HHMM < HUS2_AS01_TK01_HHMM1)), _iMAN := HUS2_AS01_TK01_MAN, _iLM_Delay := HUS2_AS01_TK01_FLM);
HUS2_AS01_TK01_IT := AUTO_MAN._bStart;
HUS2_AS01_TK01_LM := AUTO_MAN._bLM_DELAYED;
END_PROGRAM

(* POU SYSTEM/HUS2_AS01_UPPSTART, CFC *)
PROGRAM HUS2_AS01_UPPSTART
VAR

	START   :BOOL;

	START_VS1: BOOL;
	START_VS20: BOOL;
	START_VS30: BOOL;
	START_VS40: BOOL;

	On_Delay1: TON;
	On_Delay2: TON;
	On_Delay3: TON;
	On_Delay4: TON;

	On_Delay5: TON;
	On_Delay6: TON;
	On_Delay7: TON;
	START_FA1XX: BOOL;
	START_FA2XX: BOOL;
	START_FA3XX: BOOL;
END_VAR
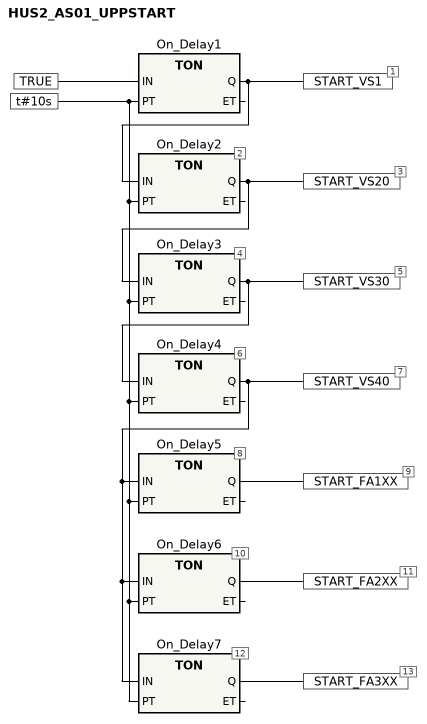
_CFC_ (* Continuous Function Chart, elements in execution order *)
#0 On_Delay1:TON(IN: TRUE, PT: t#10s)
#1 START_VS1 <= #0.Q
#2 On_Delay2:TON(IN: #0.Q, PT: t#10s)
#3 START_VS20 <= #2.Q
#4 On_Delay3:TON(IN: #2.Q, PT: t#10s)
#5 START_VS30 <= #4.Q
#6 On_Delay4:TON(IN: #4.Q, PT: t#10s)
#7 START_VS40 <= #6.Q
#8 On_Delay5:TON(IN: #6.Q, PT: t#10s)
#9 START_FA1XX <= #8.Q
#10 On_Delay6:TON(IN: #6.Q, PT: t#10s)
#11 START_FA2XX <= #10.Q
#12 On_Delay7:TON(IN: #6.Q, PT: t#10s)
#13 START_FA3XX <= #12.Q
_END_CFC_
(* the same logic as Structured Text *)
On_Delay1(IN := TRUE, PT := t#10s);
START_VS1 := On_Delay1.Q;
On_Delay2(IN := On_Delay1.Q, PT := t#10s);
START_VS20 := On_Delay2.Q;
On_Delay3(IN := On_Delay2.Q, PT := t#10s);
START_VS30 := On_Delay3.Q;
On_Delay4(IN := On_Delay3.Q, PT := t#10s);
START_VS40 := On_Delay4.Q;
On_Delay5(IN := On_Delay4.Q, PT := t#10s);
START_FA1XX := On_Delay5.Q;
On_Delay6(IN := On_Delay4.Q, PT := t#10s);
START_FA2XX := On_Delay6.Q;
On_Delay7(IN := On_Delay4.Q, PT := t#10s);
START_FA3XX := On_Delay7.Q;
END_PROGRAM

(* POU SYSTEM/Brandspjäll/AS01_BRANDSPJALL, CFC *)
PROGRAM AS01_BRANDSPJALL
VAR


END_VAR
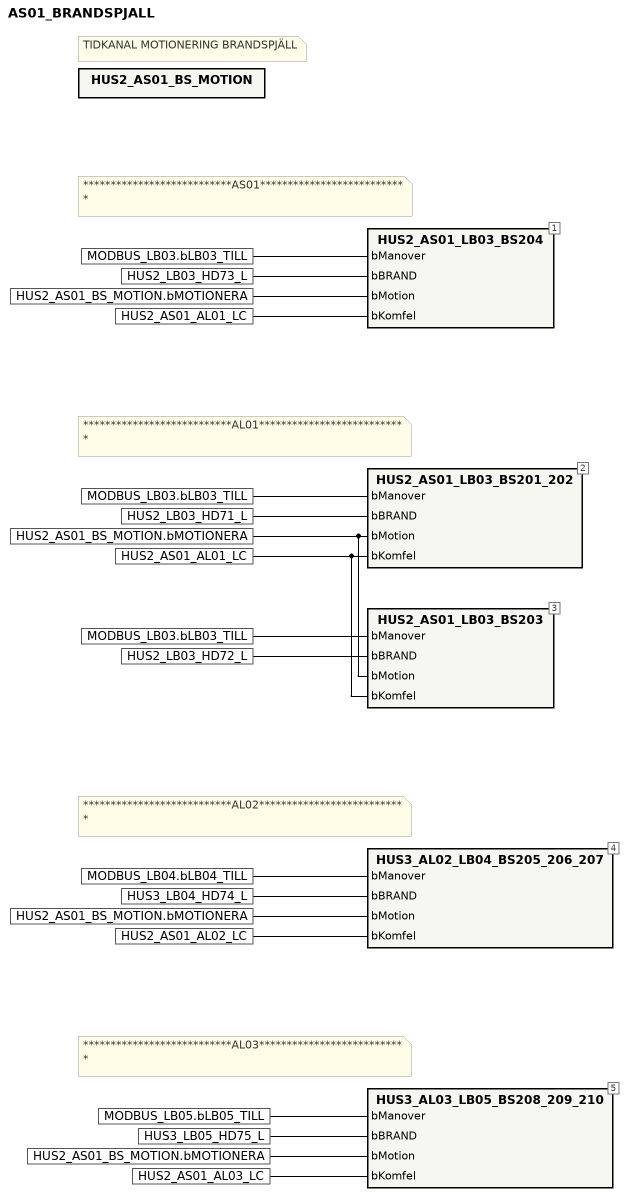
_CFC_ (* Continuous Function Chart, elements in execution order *)
(* ***************************AL03*************************** *)
(* ***************************AL02*************************** *)
(* TIDKANAL MOTIONERING BRANDSPJÄLL *)
(* ***************************AS01*************************** *)
(* ***************************AL01*************************** *)
#0 HUS2_AS01_BS_MOTION()
#1 HUS2_AS01_LB03_BS204(bManover: MODBUS_LB03.bLB03_TILL, bBRAND: HUS2_LB03_HD73_L, bMotion: HUS2_AS01_BS_MOTION.bMOTIONERA, bKomfel: HUS2_AS01_AL01_LC)
#2 HUS2_AS01_LB03_BS201_202(bManover: MODBUS_LB03.bLB03_TILL, bBRAND: HUS2_LB03_HD71_L, bMotion: HUS2_AS01_BS_MOTION.bMOTIONERA, bKomfel: HUS2_AS01_AL01_LC)
#3 HUS2_AS01_LB03_BS203(bManover: MODBUS_LB03.bLB03_TILL, bBRAND: HUS2_LB03_HD72_L, bMotion: HUS2_AS01_BS_MOTION.bMOTIONERA, bKomfel: HUS2_AS01_AL01_LC)
#4 HUS3_AL02_LB04_BS205_206_207(bManover: MODBUS_LB04.bLB04_TILL, bBRAND: HUS3_LB04_HD74_L, bMotion: HUS2_AS01_BS_MOTION.bMOTIONERA, bKomfel: HUS2_AS01_AL02_LC)
#5 HUS3_AL03_LB05_BS208_209_210(bManover: MODBUS_LB05.bLB05_TILL, bBRAND: HUS3_LB05_HD75_L, bMotion: HUS2_AS01_BS_MOTION.bMOTIONERA, bKomfel: HUS2_AS01_AL03_LC)
_END_CFC_
(* the same logic as Structured Text *)
(* ***************************AL03*************************** *)
(* ***************************AL02*************************** *)
(* TIDKANAL MOTIONERING BRANDSPJÄLL *)
(* ***************************AS01*************************** *)
(* ***************************AL01*************************** *)
HUS2_AS01_BS_MOTION();
HUS2_AS01_LB03_BS204(bManover := MODBUS_LB03.bLB03_TILL, bBRAND := HUS2_LB03_HD73_L, bMotion := HUS2_AS01_BS_MOTION.bMOTIONERA, bKomfel := HUS2_AS01_AL01_LC);
HUS2_AS01_LB03_BS201_202(bManover := MODBUS_LB03.bLB03_TILL, bBRAND := HUS2_LB03_HD71_L, bMotion := HUS2_AS01_BS_MOTION.bMOTIONERA, bKomfel := HUS2_AS01_AL01_LC);
HUS2_AS01_LB03_BS203(bManover := MODBUS_LB03.bLB03_TILL, bBRAND := HUS2_LB03_HD72_L, bMotion := HUS2_AS01_BS_MOTION.bMOTIONERA, bKomfel := HUS2_AS01_AL01_LC);
HUS3_AL02_LB04_BS205_206_207(bManover := MODBUS_LB04.bLB04_TILL, bBRAND := HUS3_LB04_HD74_L, bMotion := HUS2_AS01_BS_MOTION.bMOTIONERA, bKomfel := HUS2_AS01_AL02_LC);
HUS3_AL03_LB05_BS208_209_210(bManover := MODBUS_LB05.bLB05_TILL, bBRAND := HUS3_LB05_HD75_L, bMotion := HUS2_AS01_BS_MOTION.bMOTIONERA, bKomfel := HUS2_AS01_AL03_LC);
END_PROGRAM

(* POU SYSTEM/Brandspjäll/Tidkanal motionering/HUS2_AS01_BS_MOTION, CFC *)
PROGRAM HUS2_AS01_BS_MOTION

VAR
	AUTO_MAN: fbManualOverride;

	bMOTIONERA: BOOL;
	OffDelayMotion: TOF;
	R_RIGGA: R_TRIG;
END_VAR
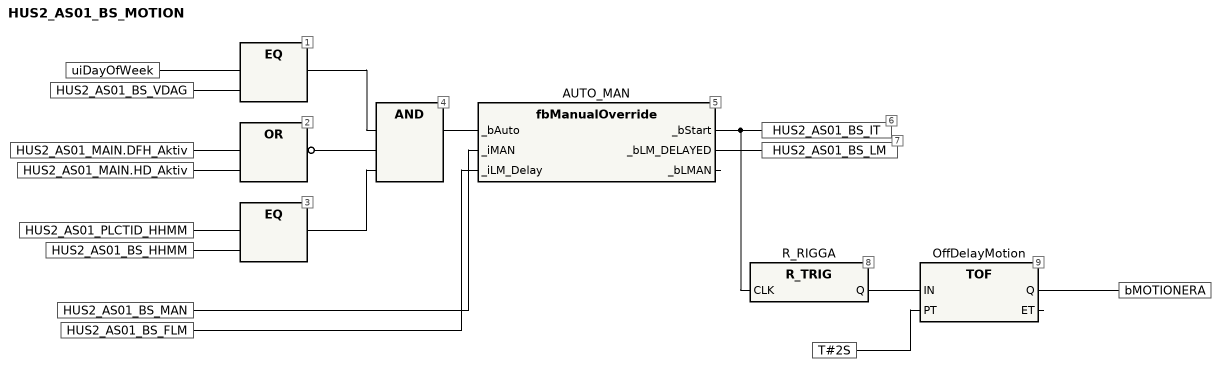
_CFC_ (* Continuous Function Chart, elements in execution order *)
#0 bMOTIONERA <= #9.Q
#1 EQ(uiDayOfWeek, HUS2_AS01_BS_VDAG)
#2 OR(HUS2_AS01_MAIN.DFH_Aktiv, HUS2_AS01_MAIN.HD_Aktiv)
#3 EQ(HUS2_AS01_PLCTID_HHMM, HUS2_AS01_BS_HHMM)
#4 AND(#1, NOT #2, #3)
#5 AUTO_MAN:fbManualOverride(_bAuto: #4, _iMAN: HUS2_AS01_BS_MAN, _iLM_Delay: HUS2_AS01_BS_FLM)
#6 HUS2_AS01_BS_IT <= #5._bStart
#7 HUS2_AS01_BS_LM <= #5._bLM_DELAYED
#8 R_RIGGA:R_TRIG(CLK: #5._bStart)
#9 OffDelayMotion:TOF(IN: #8.Q, PT: T#2S)
_END_CFC_
(* the same logic as Structured Text *)
bMOTIONERA := OffDelayMotion.Q;
AUTO_MAN(_bAuto := (uiDayOfWeek = HUS2_AS01_BS_VDAG) AND NOT (HUS2_AS01_MAIN.DFH_Aktiv OR HUS2_AS01_MAIN.HD_Aktiv) AND (HUS2_AS01_PLCTID_HHMM = HUS2_AS01_BS_HHMM), _iMAN := HUS2_AS01_BS_MAN, _iLM_Delay := HUS2_AS01_BS_FLM);
HUS2_AS01_BS_IT := AUTO_MAN._bStart;
HUS2_AS01_BS_LM := AUTO_MAN._bLM_DELAYED;
R_RIGGA(CLK := AUTO_MAN._bStart);
OffDelayMotion(IN := R_RIGGA.Q, PT := T#2S);
END_PROGRAM

(* POU SYSTEM/Brandspjäll/HD73_BS204/HUS2_AS01_LB03_BS204, FAI *)
PROGRAM HUS2_AS01_LB03_BS204

VAR_INPUT
	bManover	 	:BOOL;
	bBRAND		:BOOL;
	bMotion		:BOOL;
	bKomfel		:BOOL;
END_VAR

VAR
	_bSetDefaultLocal: BOOL;

	SetAlarmDelay: FB_HVACPersistent_Int;
	SetAlarmDelay2: FB_HVACPersistent_Int;

	SpjallStyr: fbBrandspjallStyr;

	ResetACK: fbBool_Reset;
END_VAR
(* body not read: cfc116 *)
END_PROGRAM

(* POU xEgna Funktionsblock/fbBrandspjallStyr, CFC *)
FUNCTION_BLOCK fbBrandspjallStyr
VAR_INPUT
	bManover					:BOOL;
	iMAN_Hand				:INT;
	iMAN_FL					:INT;
	bBS_IO					:BOOL;
	iBS_IO_FL					:INT;
	bBS_IS					:BOOL;
	iBS_IS_FL					:INT;
	bBRAND					:BOOL;
	bKomfel					:BOOL;
	iKomfel_FL				:INT;
	bMotion					:BOOL;
	bACK						:BOOL;

END_VAR


VAR_OUTPUT
	bManoverUt				:BOOL;
	bMotionAktiv				:BOOL;
	bLM						:BOOL;
	bFellageOppnarEJ			:BOOL;
	bFellageStangerEJ			:BOOL;
	bFellageOppetStangt		:BOOL;

END_VAR

VAR

	BrytManover: BOOL;
	MotionManover: BOOL;
	StartaMotionOppetSpjall: BOOL;
	StartaMotionStangtSpjall: BOOL;
	bResetFellage: BOOL;
	bAvslutaMot: BOOL;

	OVERRIDE: fbManualOverride;
	ResetMAN: fbAutoResetMAN;
	PulsaMotionsKommando: TP;
	DelayResetMotion: TON;

	DELAY1: fbDelayedAlarmMinutes;
	DELAY2: fbDelayedAlarmSeconds;
	DELAY3: fbDelayedAlarmSeconds;

	SETRES1: RS;
	SETRES2: RS;
	SETRES3: RS;

	Motion_oppet: RS;
	Motion_oppet_bryt: SR;
	DelayMotOppet: TON;
	Trig_bryt_man: R_TRIG;
	DelayResetMotOppet: TON;

	Motion_stangt: RS;
	Motion_stangt_manover: SR;
	DelayMotStangt: TON;
	Trig_man: R_TRIG;
	DelayResetMotStangt: TON;


END_VAR
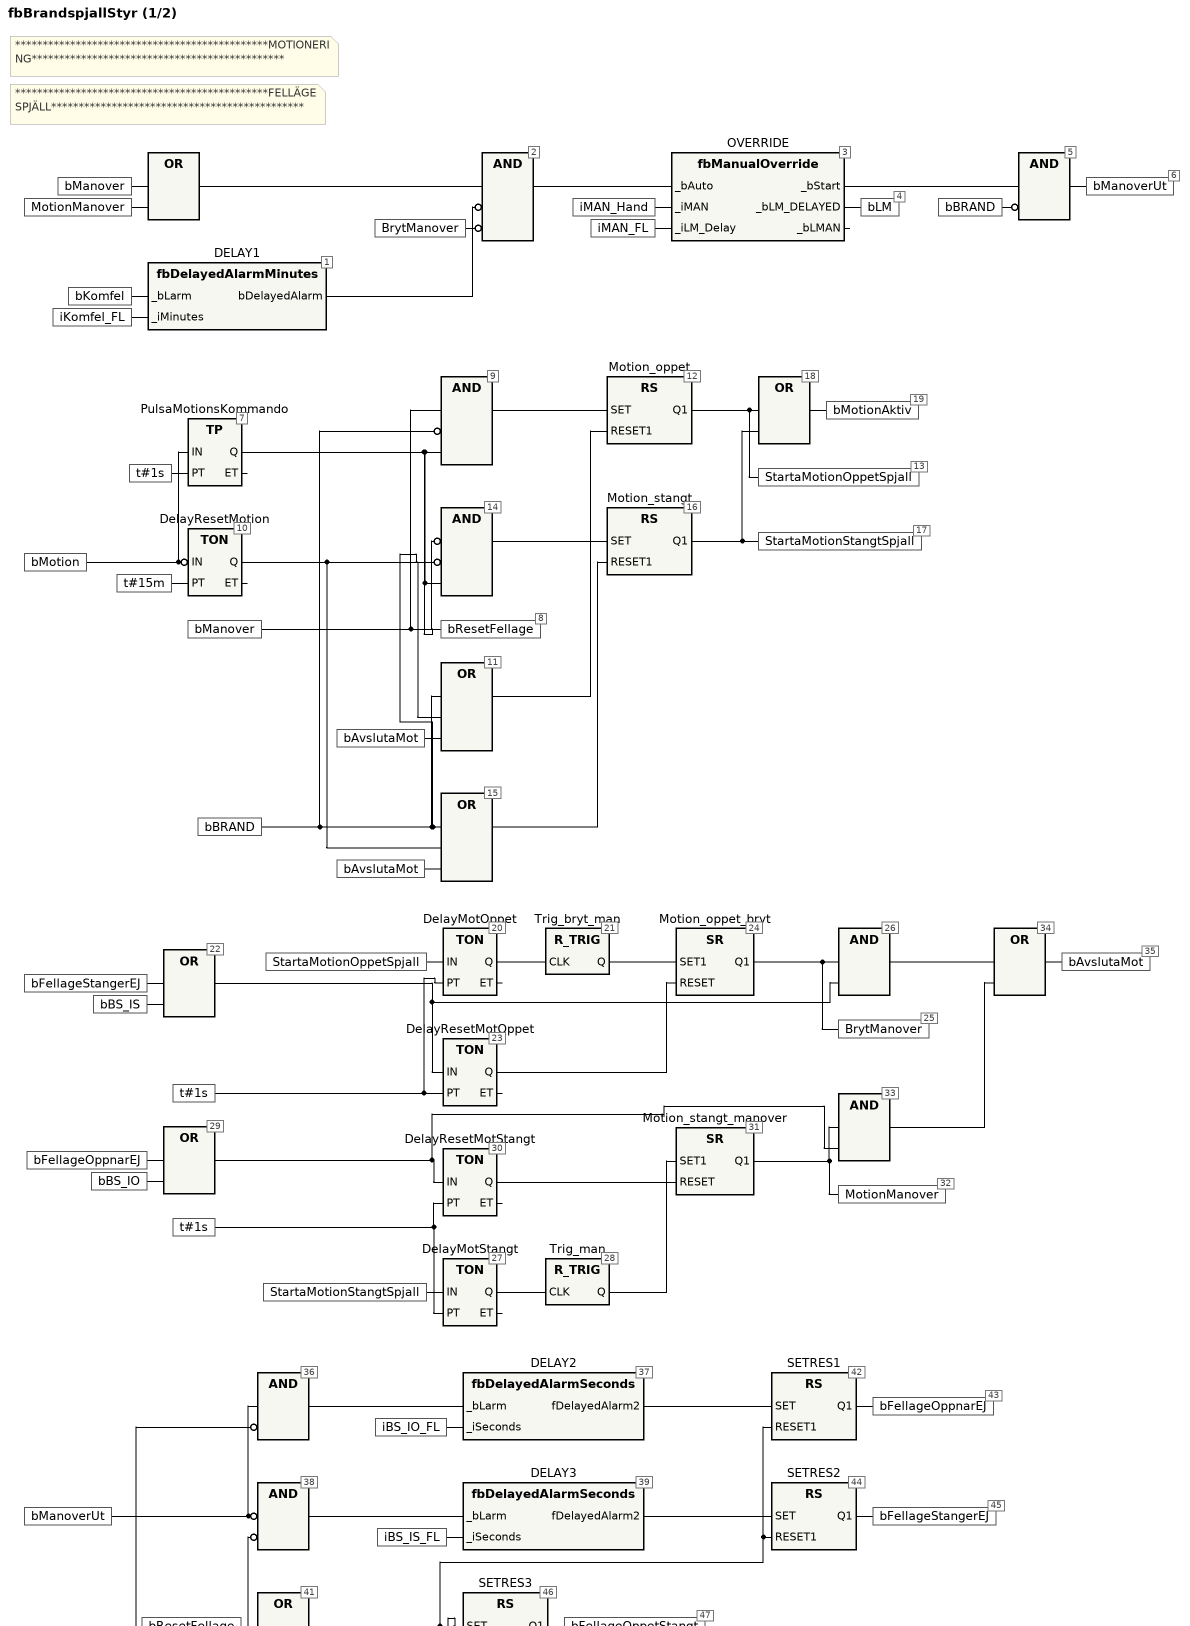
